{attribute 'qualified_only'}
{attribute 'to_string'}
TYPE ActuatorHorizontalListenerStep :
(
  Undefined := 0
  
  ,PreMoveStepBegin
  ,PreMoveStepCheckAxisVerticalPosition
  ,PreMoveStepSwitchOnLight
  ,PreMoveStepEnd
);
END_TYPE

(* stored: Version 1.1.0.1
   DUT ActuatorHorizontalListenerStep: Id {ee7095a2-52e7-469a-ac24-e4fd1ce17783} *)
